// TIA Portal V18 export
VAR_GLOBAL   // PLC tag table "Default tag table"
   FlowOn AT %Q0.1 : Bool;
   RemoteOnCommand AT %I0.1 : Bool;
END_VAR
